// TwinCAT 3 PLC project plkV2
// ProgramVersion: 3.1.4024.0
// libraries:
//   Tc2_Standard, * (Beckhoff Automation GmbH)
//   Tc2_System, * (Beckhoff Automation GmbH)
//   Tc3_Module, * (Beckhoff Automation GmbH)
// project tree:
//   AUTOmovement/ A1.TcPOU, grab.TcPOU, moveCCW.TcPOU, moveCW.TcPOU, moveDown.TcPOU, moveIN.TcPOU, moveOUT.TcPOU, moveUP.TcPOU, relise.TcPOU
//   EdgeDetection/ EdgeDetection.TcPOU
//   / getBreadFromSensors.TcPOU, PlcTask.TcTTO
//   GVLs/ GVL.TcGVL, HMI.TcGVL
//   Muliplex/ Multiplexer.TcPOU
//   POUs/Automatic/ Automatic.TcPOU, AutomaticFB.TcPOU, FirstMove.TcPOU, SortTest.TcPOU, startSorting.TcPOU
//   POUs/ MAIN.TcPOU, MasterControl.TcPOU
//   POUs/Manual/ Manual.TcPOU
//   Timer/ AUTOtimer.TcPOU, TIMER.TcPOU

CONFIGURATION plkV2
    RESOURCE PLC ON TwinCAT3
        TASK PlcTask(INTERVAL := T#10ms, PRIORITY := 20);
        PROGRAM MasterControl WITH PlcTask : MasterControl;
    END_RESOURCE
END_CONFIGURATION

// ---- GVLs/GVL.TcGVL
{attribute 'qualified_only'}
VAR_GLOBAL
	//Automatic/manual
	ToggleSwitch AT %I* : BOOL; //0 - automatic; 1 - manual
	
	//lights
	LEDRed AT %Q* : BOOL; 
	LEDGreen AT %Q* : BOOL; 
	LEDupperBlue AT %Q* : BOOL; 
	LEDdownBlue AT %Q* : BOOL; 
	
	//buttons
	//upper
	ULBButton AT %I* : BOOL;
	URBButton AT %I* : BOOL;
	//lover
	LLBButton AT %I* : BOOL;
	LRBButton AT %I* : BOOL;
	//color
	GButton AT %I* : BOOL;
	RButton AT %I* : BOOL;


	//MOVESET
	//MoveUp/Down
	riseWay AT %Q* : BOOL; //0 - down, 1 - up
	riseAction AT %Q* : BOOL;
	
	
	//Rotation
	rotationWay AT %Q* : BOOL; //0 - CW, 1 - CCW
	rotationAction AT %Q* : BOOL;
	
	
	//Stretch
	stretchWay AT %Q* : BOOL; //0 - stretch, 1 - shrink
	stretchAction AT %Q* : BOOL;
	
	//claw
	clawWay AT %Q* : BOOL; //0 - open, 1 - release
	clawAction AT %Q* : BOOL;
	
	
	//SWITCHES
	//rotation
	SWrotation AT %I* : BOOL;
	SWstepsRotation AT %I* : BOOL;
	
	//stretch
	SWstretch AT %I* : BOOL;
	SWstepsStretch AT %I* : BOOL;
	
	//rise
	SWrise AT %I* : BOOL;
	SWstepsRise AT %I* : BOOL;
	
	//grab
	SWgrab AT %I* : BOOL;
	SWstepsGrab AT %I* : BOOL;
	
	
	//Bakery
	weight: REAL; //light - bagel, medium - toast/rye, heavy - baguette (weight sensor - HX711)
	color: INT; //white/black (color sensor - TCS3472)
	breadType: INT; //toast = 0; baguette = 1; rye = 2; bagel = 3
	binNumber: INT; // 2 or 4
	binFull: BOOL; //HC-SR04 x 2 or 4
	breadInfo : STRING; // white toast, white beguette, dark rye, dark bagel
	
	//objekt za pekarno - za HMI
	{attribute 'TcHmiSymbol'}
	BreadInfoID : INT := 0;
	
	
	{attribute 'TcHmiSymbol'}
	BinFullNumber : INT := 0;
	
	
	//nove lastnosti za senzorje
	breadColor : INT;
    breadWeightClass : STRING(10);
	breadID: INT;
	
 	{attribute 'TcHmiSymbol'}
	breadIDinfo : INT := 0;
	{attribute 'TcHmiSymbol'}
	breadIDText : STRING(10) := '';

    fullBin : INT;
	
	
	//za posodabljat koliko elementov je v škatli
	{attribute 'TcHmiSymbol'}
	BinUpdateTrigger : INT := 0;
	
	
	{attribute 'TcHmiSymbol'}
	breadTypeImageID : INT := 0; // 0=none, 1=toast, 2=baguette, 3=rye, 4=bagel
	//Sensors
	//BinIsFull : BOOL := FALSE;
	BinIsFull : INT := 0;	
	{attribute 'TcHmiSymbol'} Bin1Full : BOOL := FALSE;
	{attribute 'TcHmiSymbol'} Bin2Full : BOOL := FALSE;
	{attribute 'TcHmiSymbol'} Bin3Full : BOOL := FALSE;
	{attribute 'TcHmiSymbol'} Bin4Full : BOOL := FALSE;
	
	//breadColor: white, black
	{attribute 'TcHmiSymbol'}
	//breadColor : STRING(10) := 'NONE';
	
	
	//Number of bread in bin
    numToast   : INT := 0;
    numBaguette: INT := 0;
    numRye     : INT := 0;
    numBagel   : INT := 0;
	
	//STEVCI
	UniversalStevec AT %I* : BOOL;
	stevecGor AT %I* : BOOL;
	stevecRotacija AT %I* : BOOL;
	stevecSkrci AT %I* : BOOL;
	stevecKlesce AT %I* : BOOL;
	
	height AT %I* : REAL;
	rotation AT %I* : REAL;
	length AT %I* : REAL;
	grabMeter AT %I* : REAL;
	
	
	// AVTOMATIK PREMIKI
	upDone AT %Q* : BOOL;
	downDone AT %Q* : BOOL;
	CWDone AT %Q* : BOOL;
	CCWDone AT %Q* : BOOL;
	skrciDone AT %Q* : BOOL;
	raztegniDone AT %Q* : BOOL;
	grabDone AT %Q* : BOOL;
	reliseDone AT %Q* : BOOL;
	
	//GOR DOL
	gor AT %Q* : BOOL;
	dol AT %Q* : BOOL;
	
	//LEVO DESNO
	CW AT %Q* : BOOL;
	CCW AT %Q* : BOOL;
	
	//KLEŠČE--NE DELA!!!!
	primi AT %Q* : BOOL;
	spusti AT %Q* : BOOL;
	
	//IZTEG--NE DELA!!!!
	raztegniNaprej AT %Q* : BOOL;
	skrci AT %Q* : BOOL;
	
	
	//on/off
	isON AT %I* : BOOL;
END_VAR

// ---- GVLs/HMI.TcGVL
{attribute 'qualified_only'}
VAR_GLOBAL
	BreadIDpicked:INT;
	test:BOOL := FALSE;
	Action1:BOOL;
	Action2:BOOL;
END_VAR

// ---- POUs/MasterControl.TcPOU
PROGRAM MasterControl
VAR
	//preveri če je switvh aktiven
	Rocno: Manual;
	Avtomatik: Automatic;
	{attribute 'TcHmiSymbol'}
	premikanje: SortTest;

	
	
	Motor: BOOL;
	IS_Manual: BOOL;
	
	// Nova instanca za vrednotenje kruha
	BreadEval: getBreadFromSensors;
	
END_VAR

IS_Manual := GVL.ToggleSwitch;
IF IS_Manual THEN
	Rocno();
	//GVL.riseWay := Rocno.smer1;//asign GVL.way
ELSE
		//Avtomatik();
		premikanje();
END_IF

// Neodvisno od ročnega/avtomatskega režima – vedno preveri kruh
BreadEval(
	breadColor := GVL.breadColor,
	breadWeightClass := GVL.breadWeightClass
);

// Rezultat zapiši v GVL za HMI uporabo
GVL.breadTypeImageID := BreadEval.breadTypeImageID;
GVL.breadInfo := BreadEval.breadInfo;

END_PROGRAM

// ---- POUs/Manual/Manual.TcPOU
FUNCTION_BLOCK Manual
VAR_INPUT
END_VAR

VAR_OUTPUT
END_VAR

VAR
	motorSelect: Multiplexer;
	EdgeDetectionRedButton: EdgeDetection;
	TIMER: TIMER;
	
	CountDown: CTUD;
	EdgeDetectionCD: BOOL;
	dropTimer: TON;
	rotateTimer: TON;
	stretchTimer: TON;
	clawTimer: TON;
	CounterDol: CTUD;
	visina: WORD;
	CounterCCW: CTUD;
	rotacija: WORD;
	CounterRazteg: CTUD;
	dolzina: WORD;
	CounterKlesce: CTUD;
	prijem: WORD;
	CounterVisina: CTUD;
END_VAR

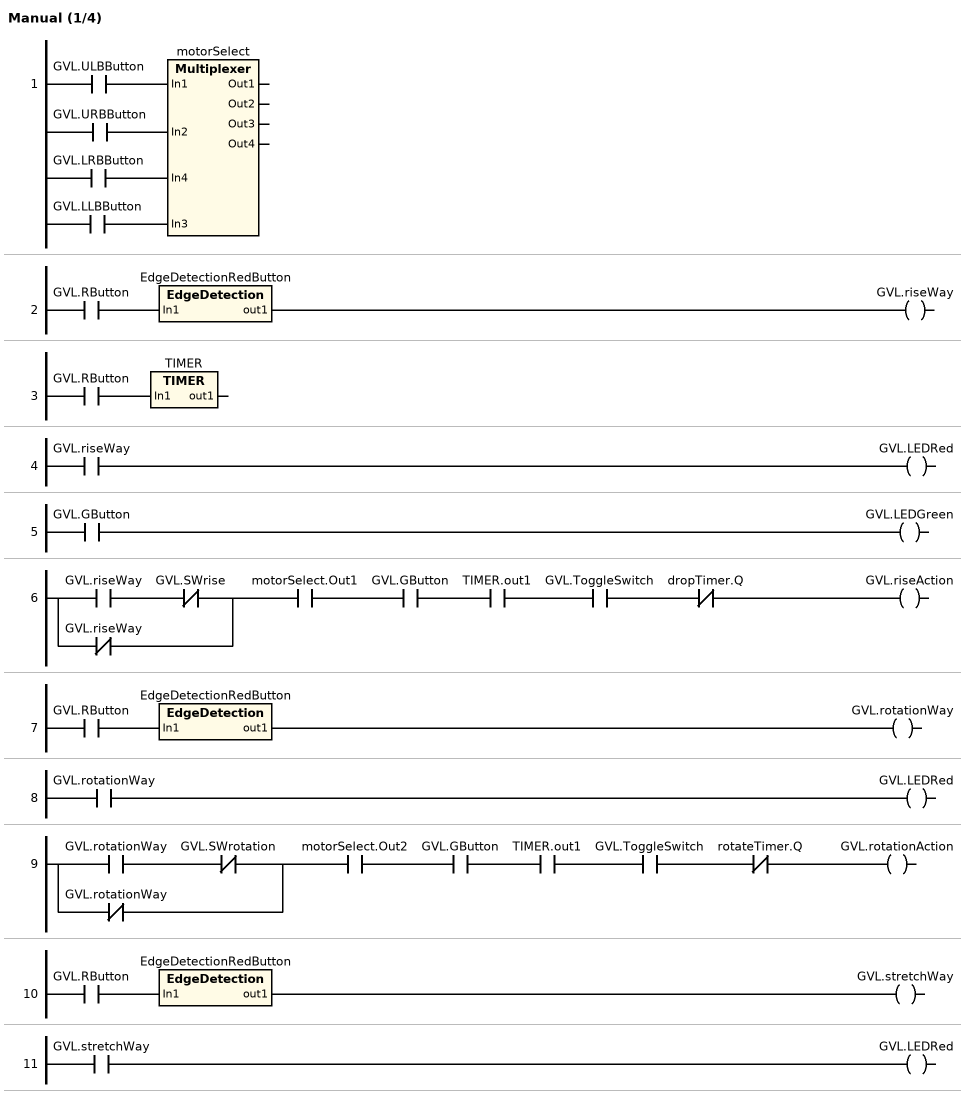
// NETWORK 1
motorSelect(In1 := GVL.ULBButton, In2 := GVL.URBButton, In4 := GVL.LRBButton, In3 := GVL.LLBButton); // Multiplexer

// NETWORK 2
EdgeDetectionRedButton(In1 := GVL.RButton); // EdgeDetection
GVL.riseWay := EdgeDetectionRedButton.out1;

// NETWORK 3
TIMER(In1 := GVL.RButton);

// NETWORK 4
GVL.LEDRed := GVL.riseWay;

// NETWORK 5
GVL.LEDGreen := GVL.GButton;

// NETWORK 6
GVL.riseAction := (GVL.riseWay AND NOT GVL.SWrise OR NOT GVL.riseWay) AND motorSelect.Out1 AND GVL.GButton AND TIMER.out1 AND GVL.ToggleSwitch AND NOT dropTimer.Q;

// NETWORK 7
EdgeDetectionRedButton(In1 := GVL.RButton); // EdgeDetection
GVL.rotationWay := EdgeDetectionRedButton.out1;

// NETWORK 8
GVL.LEDRed := GVL.rotationWay;

// NETWORK 9
GVL.rotationAction := (GVL.rotationWay AND NOT GVL.SWrotation OR NOT GVL.rotationWay) AND motorSelect.Out2 AND GVL.GButton AND TIMER.out1 AND GVL.ToggleSwitch AND NOT rotateTimer.Q;

// NETWORK 10
EdgeDetectionRedButton(In1 := GVL.RButton); // EdgeDetection
GVL.stretchWay := EdgeDetectionRedButton.out1;

// NETWORK 11
GVL.LEDRed := GVL.stretchWay;

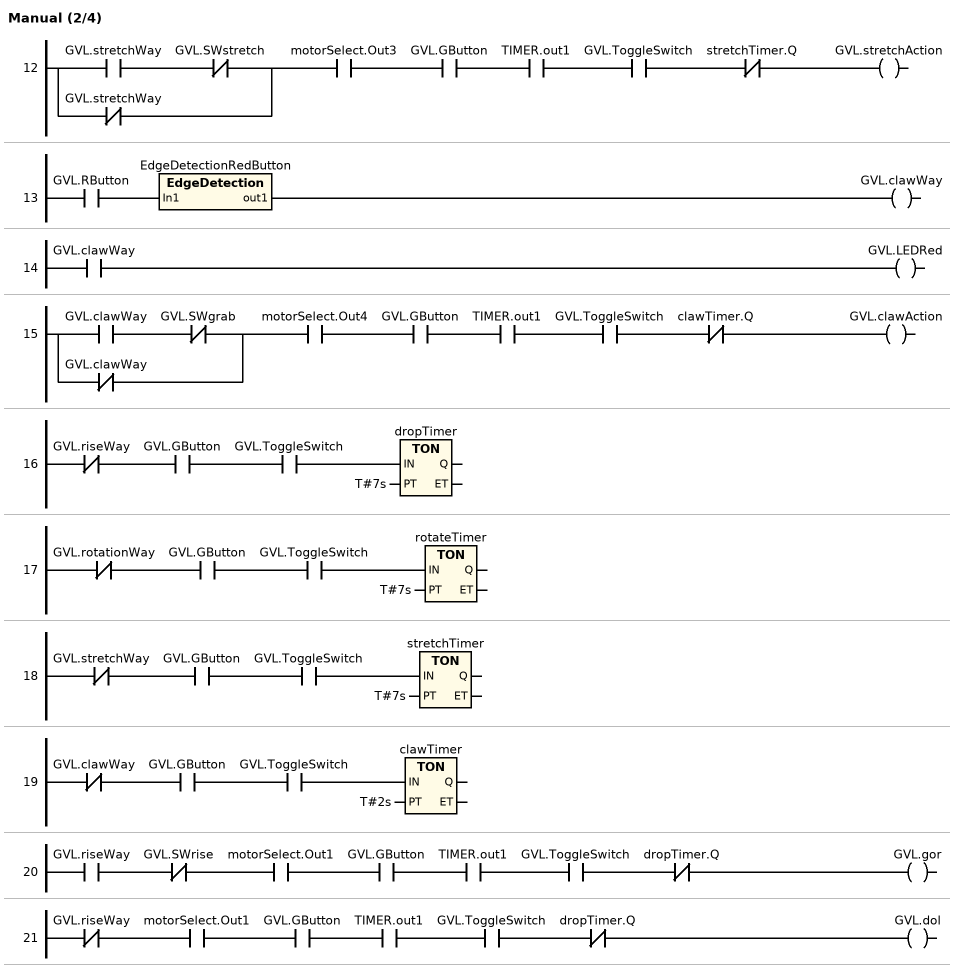
// NETWORK 12
GVL.stretchAction := (GVL.stretchWay AND NOT GVL.SWstretch OR NOT GVL.stretchWay) AND motorSelect.Out3 AND GVL.GButton AND TIMER.out1 AND GVL.ToggleSwitch AND NOT stretchTimer.Q;

// NETWORK 13
EdgeDetectionRedButton(In1 := GVL.RButton); // EdgeDetection
GVL.clawWay := EdgeDetectionRedButton.out1;

// NETWORK 14
GVL.LEDRed := GVL.clawWay;

// NETWORK 15
GVL.clawAction := (GVL.clawWay AND NOT GVL.SWgrab OR NOT GVL.clawWay) AND motorSelect.Out4 AND GVL.GButton AND TIMER.out1 AND GVL.ToggleSwitch AND NOT clawTimer.Q;

// NETWORK 16
dropTimer(IN := NOT GVL.riseWay AND GVL.GButton AND GVL.ToggleSwitch, PT := T#7s); // TON

// NETWORK 17
rotateTimer(IN := NOT GVL.rotationWay AND GVL.GButton AND GVL.ToggleSwitch, PT := T#7s); // TON

// NETWORK 18
stretchTimer(IN := NOT GVL.stretchWay AND GVL.GButton AND GVL.ToggleSwitch, PT := T#7s); // TON

// NETWORK 19
clawTimer(IN := NOT GVL.clawWay AND GVL.GButton AND GVL.ToggleSwitch, PT := T#2s); // TON

// NETWORK 20
GVL.gor := GVL.riseWay AND NOT GVL.SWrise AND motorSelect.Out1 AND GVL.GButton AND TIMER.out1 AND GVL.ToggleSwitch AND NOT dropTimer.Q;

// NETWORK 21
GVL.dol := NOT GVL.riseWay AND motorSelect.Out1 AND GVL.GButton AND TIMER.out1 AND GVL.ToggleSwitch AND NOT dropTimer.Q;

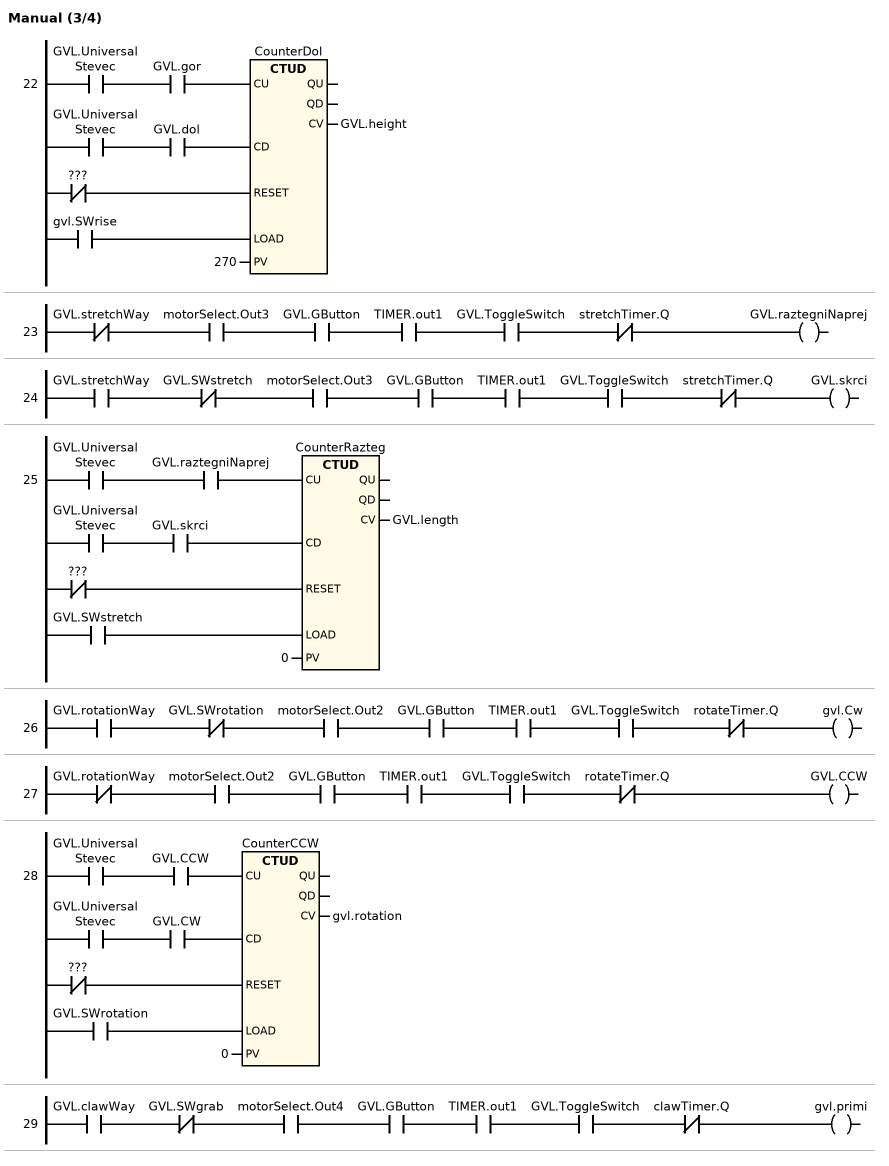
// NETWORK 22
CounterDol(
    CU := GVL.UniversalStevec AND GVL.gor,
    CD := GVL.UniversalStevec AND GVL.dol,
    LOAD := gvl.SWrise,
    PV := 270,
    CV => GVL.height); // CTUD

// NETWORK 23
GVL.raztegniNaprej := NOT GVL.stretchWay AND motorSelect.Out3 AND GVL.GButton AND TIMER.out1 AND GVL.ToggleSwitch AND NOT stretchTimer.Q;

// NETWORK 24
GVL.skrci := GVL.stretchWay AND NOT GVL.SWstretch AND motorSelect.Out3 AND GVL.GButton AND TIMER.out1 AND GVL.ToggleSwitch AND NOT stretchTimer.Q;

// NETWORK 25
CounterRazteg(
    CU := GVL.UniversalStevec AND GVL.raztegniNaprej,
    CD := GVL.UniversalStevec AND GVL.skrci,
    LOAD := GVL.SWstretch,
    PV := 0,
    CV => GVL.length); // CTUD

// NETWORK 26
gvl.Cw := GVL.rotationWay AND NOT GVL.SWrotation AND motorSelect.Out2 AND GVL.GButton AND TIMER.out1 AND GVL.ToggleSwitch AND NOT rotateTimer.Q;

// NETWORK 27
GVL.CCW := NOT GVL.rotationWay AND motorSelect.Out2 AND GVL.GButton AND TIMER.out1 AND GVL.ToggleSwitch AND NOT rotateTimer.Q;

// NETWORK 28
CounterCCW(
    CU := GVL.UniversalStevec AND GVL.CCW,
    CD := GVL.UniversalStevec AND GVL.CW,
    LOAD := GVL.SWrotation,
    PV := 0,
    CV => gvl.rotation); // CTUD

// NETWORK 29
gvl.primi := GVL.clawWay AND NOT GVL.SWgrab AND motorSelect.Out4 AND GVL.GButton AND TIMER.out1 AND GVL.ToggleSwitch AND NOT clawTimer.Q;

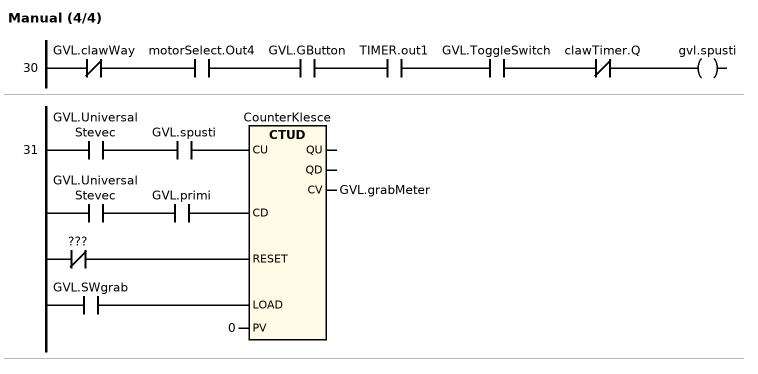
// NETWORK 30
gvl.spusti := NOT GVL.clawWay AND motorSelect.Out4 AND GVL.GButton AND TIMER.out1 AND GVL.ToggleSwitch AND NOT clawTimer.Q;

// NETWORK 31
CounterKlesce(
    CU := GVL.UniversalStevec AND GVL.spusti,
    CD := GVL.UniversalStevec AND GVL.primi,
    LOAD := GVL.SWgrab,
    PV := 0,
    CV => GVL.grabMeter); // CTUD

END_FUNCTION_BLOCK

// ---- Muliplex/Multiplexer.TcPOU
FUNCTION_BLOCK Multiplexer
VAR_INPUT
	In1: BOOL;
	In2: BOOL;
	In4: BOOL;
	In3: BOOL;
END_VAR

VAR_OUTPUT
	Out1: BOOL;
	Out2: BOOL;
	Out3: BOOL;
	Out4: BOOL;
END_VAR

VAR
	UpDown: RS;
	CWCCW: RS;
	StretchShrink: RS;
	GrabRelease: RS;
END_VAR

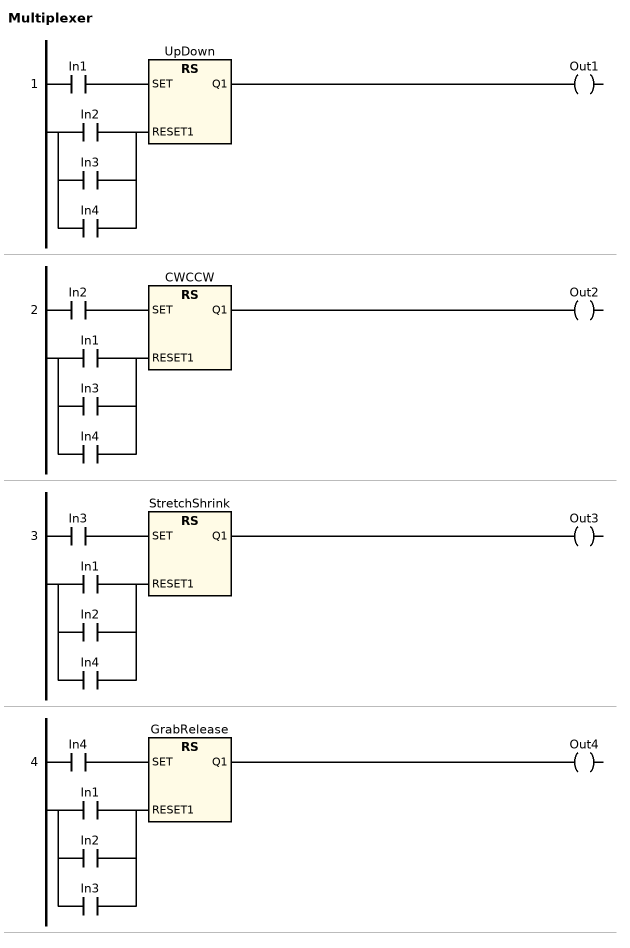
// NETWORK 1
UpDown(SET := In1, RESET1 := In2 OR In3 OR In4); // RS
Out1 := UpDown.Q1;

// NETWORK 2
CWCCW(SET := In2, RESET1 := In1 OR In3 OR In4); // RS
Out2 := CWCCW.Q1;

// NETWORK 3
StretchShrink(SET := In3, RESET1 := In1 OR In2 OR In4); // RS
Out3 := StretchShrink.Q1;

// NETWORK 4
GrabRelease(SET := In4, RESET1 := In1 OR In2 OR In3); // RS
Out4 := GrabRelease.Q1;

END_FUNCTION_BLOCK

// ---- EdgeDetection/EdgeDetection.TcPOU
FUNCTION_BLOCK EdgeDetection
VAR_INPUT
	In1: BOOL;
END_VAR
VAR_OUTPUT
	out1: BOOL;
END_VAR
VAR
	EdgeDetection1: R_TRIG;
	MemoryCell1: RS;
END_VAR

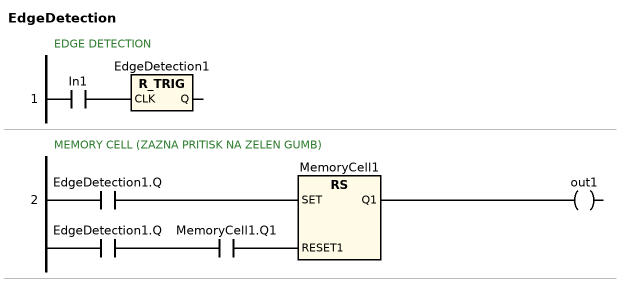
// NETWORK 1
// EDGE DETECTION
EdgeDetection1(CLK := In1); // R_TRIG

// NETWORK 2
// MEMORY CELL (ZAZNA PRITISK NA ZELEN GUMB)
MemoryCell1(SET := EdgeDetection1.Q, RESET1 := EdgeDetection1.Q AND MemoryCell1.Q1); // RS
out1 := MemoryCell1.Q1;

END_FUNCTION_BLOCK

// ---- Timer/TIMER.TcPOU
FUNCTION_BLOCK TIMER
VAR_INPUT
	In1: BOOL;
END_VAR
VAR_OUTPUT
	out1: BOOL;
END_VAR
VAR
	Timer1: TON;
	ontValue: TIME;
END_VAR

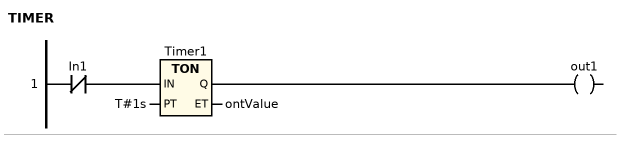
// NETWORK 1
Timer1(IN := NOT In1, PT := T#1s, ET => ontValue); // TON
out1 := Timer1.Q;

END_FUNCTION_BLOCK

// ---- POUs/Automatic/Automatic.TcPOU
FUNCTION_BLOCK Automatic
VAR_INPUT	
END_VAR
VAR_OUTPUT
END_VAR
VAR
    R1 : FirstMove;
    previousBreadID : INT := 0;
	i : INT := 1;
    triggerStart : BOOL := FALSE;
    isRunning : BOOL := FALSE;
END_VAR

// Če kruh še ni v obdelavi in pride nov breadID
//IF NOT isRunning AND GVL.breadID <> 0 AND GVL.breadID <> previousBreadID THEN
IF NOT isRunning AND GVL.breadID <> 0 THEN
	R1.itemID := GVL.breadID; // Nastavi novi kruh
	triggerStart := TRUE;
	previousBreadID := GVL.breadID; // Posodobi si trenutno vrednost
END_IF

// Poženi sekvenco, če je bil sprožen nov klic
IF triggerStart THEN
	R1(); // Pokliči FB
	isRunning := TRUE;
END_IF

// Nadaljuj izvajanje sekvence
IF isRunning THEN
	R1(); // Sekvenca se še izvaja
   IF R1.done THEN
		isRunning := FALSE;
		GVL.breadID := 0;           // Reset za TwinCAT
		previousBreadID := 0;       // Omogoči, da tudi isti kruh lahko pride ponovno
		triggerStart := FALSE;      // Reset sprožilca
	END_IF
END_IF

END_FUNCTION_BLOCK

// ---- POUs/Automatic/FirstMove.TcPOU
FUNCTION_BLOCK FirstMove
VAR_INPUT
    grab: grab; 
	timer : TP;	
	ccw: moveCCW;
	cw:moveCW;
	down:moveDown;
	iztegni:moveOUT;
	skrci:moveIN;
	up: moveUp;
	relise: relise; 
	itemID: INT := GVL.breadID;
END_VAR
VAR_OUTPUT
	 done: BOOL := FALSE; // Indikator, da je sekvenca zaključena
END_VAR
VAR
	currentState: INT := 0; // Trenutno stanje sekvence
	
	obDol: INT;
	objekt: INT;
	//itemID: INT := 1; //item number
	
	TimerWait: TOF;
	I: INT;
END_VAR

CASE currentState OF
	
	0:
		done := FALSE;
		GVL.downDone := FALSE;
		GVL.grabDone := FALSE;
		currentState := 1;
	
	1:
		down(seconds := T#5S);  // Aktiviraj premik dol
		IF GVL.downDone THEN          // Počakaj, da je premik zaključen
			currentState := 2;     // Premik na naslednje stanje
			GVL.downDone := FALSE;
		END_IF
		
	2:
		grab(seconds := T#2.2S);
		IF GVL.grabDone THEN           // Počakaj, da je prijem zaključen
			currentState := 3;      // Premik na naslednje stanje
			GVL.grabDone := FALSE;
		END_IF
		
	3:
		up(seconds := T#7S);
        IF GVL.upDone THEN           // Počakaj, da je prijem zaključen
            currentState := 4;      // Premik na naslednje stanje
			GVL.upDone := FALSE;
        END_IF

	4:
		//bageta
		IF itemID = 1 THEN
			cw(seconds := T#1.9S);
			IF GVL.CWDone THEN           // Počakaj, da je prijem zaključen
				currentState := 5;      // Premik na naslednje stanje
				GVL.CWDone := FALSE;
			END_IF
		//toast
		ELSIF itemID = 2 THEN
			cw(seconds := T#2.6S);
			IF GVL.CWDone THEN           // Počakaj, da je prijem zaključen
				currentState := 5;      // Premik na naslednje stanje
				GVL.CWDone := FALSE;
			END_IF
		//rženi kruh
		ELSIF itemID = 3 THEN
			cw(seconds := T#3.7S);
			IF GVL.CWDone THEN           // Počakaj, da je prijem zaključen
				currentState := 5;      // Premik na naslednje stanje
				GVL.CWDone := FALSE;
			END_IF
		//bagel
		ELSIF itemID = 4 THEN
			cw(seconds := T#4.2S);
			IF GVL.CWDone THEN           // Počakaj, da je prijem zaključen
				currentState := 5;      // Premik na naslednje stanje
				GVL.CWDone := FALSE;
			END_IF
		END_IF
		
	
	5:
	IF itemID = 1 THEN
		iztegni(seconds := T#4S);
        IF GVL.skrciDone THEN           // Počakaj, da je prijem zaključen
            currentState := 6;      // Premik na naslednje stanje
			GVL.skrciDone := FALSE;
        END_IF
	ELSIF itemID = 2 THEN
		iztegni(seconds := T#2.3S);
        IF GVL.skrciDone THEN           // Počakaj, da je prijem zaključen
            currentState := 6;      // Premik na naslednje stanje
			GVL.skrciDone := FALSE;
        END_IF
	ELSIF itemID = 3 THEN				
		iztegni(seconds := T#2.3S);
        IF GVL.skrciDone THEN           // Počakaj, da je prijem zaključen
            currentState := 6;      // Premik na naslednje stanje
			GVL.skrciDone := FALSE;
        END_IF
	ELSIF itemID = 4 THEN
		iztegni(seconds := T#4.3S);
        IF GVL.skrciDone THEN           // Počakaj, da je prijem zaključen
            currentState := 6;      // Premik na naslednje stanje
			GVL.skrciDone := FALSE;
        END_IF
	END_IF
		
	
	6:
		relise(seconds := T#3S);
        IF GVL.reliseDone THEN           // Počakaj, da je prijem zaključen
            currentState := 7;      // Premik na naslednje stanje
			GVL.reliseDone := FALSE;
        END_IF
	
	7:
		skrci(seconds := T#6S);
        IF GVL.skrciDone THEN           // Počakaj, da je prijem zaključen
            currentState := 8;      // Premik na naslednje stanje
			GVL.skrciDone := FALSE;
        END_IF
	
	8:
		ccw(seconds := T#6S);
        IF GVL.CWDone THEN           // Počakaj, da je prijem zaključen
            //currentState := 9;      // Premik na naslednje stanje
			currentState := 9;
			GVL.CWDone := FALSE;
        END_IF
		
	//9:
	//	GVL.upDone := FALSE;
	//	up(seconds := T#7S);
    //    IF GVL.upDone THEN           // Počakaj, da je prijem zaključen
    //        currentState := 0;      // Premik na naslednje stanje
	//		GVL.upDone := FALSE;
    //    END_IF
	
	 9:
        done := TRUE;               // Označi, da je sekvenca zaključena
        currentState := 0;          // Ponastavi na začetno stanje

	 
END_CASE

END_FUNCTION_BLOCK

// ---- AUTOmovement/grab.TcPOU
FUNCTION_BLOCK grab
VAR_INPUT
	 seconds: TIME; //time of moving	  
END_VAR
VAR_OUTPUT
	done: BOOL := FALSE; // output of finished work
END_VAR
VAR
	TimerNewGrab: AUTOtimer;
	activated: BOOL := FALSE; // Internal logic for activation
	grabEnd: BOOL := FALSE;
END_VAR

IF NOT activated THEN
    TimerNewGrab(vrednost := TRUE, inpCas := seconds, outCas => grabEnd);
    activated := TRUE;
END_IF

IF grabEnd  THEN
    TimerNewGrab(vrednost := FALSE, inpCas := seconds, outCas => grabEnd);
	GVL.primi := TRUE;
	GVL.clawWay := FALSE;
    GVL.clawAction := TRUE;  // grab active 
    GVL.grabDone := FALSE; // The move is not finished yet
	GVL.grabMeter := GVL.grabMeter + 0.4;
ELSE
	GVL.primi  := FALSE;
	GVL.clawWay := FALSE;
    GVL.clawAction := FALSE;     // Stop grabing
    GVL.grabDone:= TRUE;  // Mark the end of the move
	activated := FALSE;
END_IF

END_FUNCTION_BLOCK

// ---- Timer/AUTOtimer.TcPOU
FUNCTION_BLOCK AUTOtimer
VAR_INPUT
	vrednost: BOOL;
	inpCas: TIME;
END_VAR
VAR_OUTPUT
	outCas: BOOL;
END_VAR
VAR
	TimerAutomatic: TOF;
END_VAR

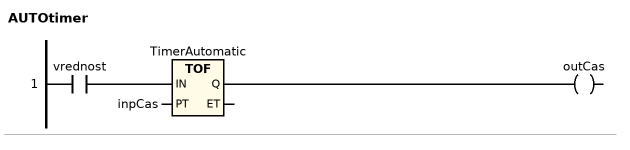
// NETWORK 1
TimerAutomatic(IN := vrednost, PT := inpCas); // TOF
outCas := TimerAutomatic.Q;

END_FUNCTION_BLOCK

// ---- AUTOmovement/moveCCW.TcPOU
FUNCTION_BLOCK moveCCW
VAR_INPUT
	 seconds: TIME;  //time of moving
END_VAR
VAR_OUTPUT
	 done: BOOL := FALSE; // output of finished work
END_VAR
VAR
	TimerNewCCW: AUTOtimer; 
	activated: BOOL := FALSE; // Internal logic for activation
	CCWend: BOOL := FALSE;
END_VAR

IF NOT activated THEN
    TimerNewCCW(vrednost := TRUE, inpCas := seconds, outCas => CCWend);
    activated := TRUE;
END_IF

IF CCWend AND NOT GVL.SWrotation THEN
    TimerNewCCW(vrednost := FALSE, inpCas := seconds, outCas => CCWend);
	GVL.CCW := TRUE;
    GVL.rotationWay := TRUE;      
	GVL.rotationAction := TRUE;  // CCW active 
  	GVL.CCWDone := FALSE;    // The move is not finished yet
	GVL.rotation := GVL.rotation - 0.5;
ELSE
	GVL.CCW := FALSE; 
   	GVL.rotationWay := FALSE;      
	GVL.rotationAction := FALSE;    // Stop moving CCW
   	GVL.CCWDone := TRUE;   // Mark the end of the move
	activated := FALSE;
END_IF

END_FUNCTION_BLOCK

// ---- AUTOmovement/moveCW.TcPOU
FUNCTION_BLOCK moveCW
VAR_INPUT
	seconds: TIME; //time of moving
END_VAR
VAR_OUTPUT
	 done: BOOL := FALSE; // output of finished work
END_VAR
VAR
	TimerNewCW: AUTOtimer;
	activated: BOOL := FALSE; // Internal logic for activation
	CWend: BOOL := FALSE;
END_VAR

IF NOT activated THEN
    TimerNewCW(vrednost := TRUE, inpCas := seconds, outCas => CWend);
    activated := TRUE;
END_IF

IF CWend THEN
    TimerNewCW(vrednost := FALSE, inpCas := seconds, outCas => CWend);
	GVL.CW := TRUE; 
    GVL.rotationWay := FALSE; 
	GVL.rotationAction := TRUE;  // CCW active 
  	GVL.CWDone := FALSE;     // The move is not finished yet
	GVL.rotation := GVL.rotation + 0.5;
ELSE
	GVL.CW := FALSE;
   	GVL.rotationWay := FALSE; 
	GVL.rotationAction := FALSE;        // Stop moving CW
    GVL.CWDone := TRUE;    // Mark the end of the move
	//CWend := FALSE;
	activated := FALSE;
END_IF

END_FUNCTION_BLOCK

// ---- AUTOmovement/moveDown.TcPOU
FUNCTION_BLOCK moveDown
VAR_INPUT
	seconds: TIME; //time of moving
END_VAR
VAR_OUTPUT
	done: BOOL := FALSE;  // output of finished work
END_VAR
VAR
	TimerNewDown: AUTOtimer; 
	aktiviran: BOOL := FALSE; // Internal logic for activation
	DownEnd: BOOL := FALSE;
END_VAR

IF NOT aktiviran THEN
    TimerNewDown(vrednost := TRUE, inpCas := seconds, outCas => DownEnd);
    aktiviran := TRUE;
END_IF

IF DownEnd THEN
    TimerNewDown(vrednost := FALSE, inpCas := seconds, outCas => DownEnd);
	GVL.dol := TRUE;
	GVL.riseWay := FALSE;
	GVL.riseAction := TRUE; 	// down active 
  	GVL.downDone := FALSE;    // The move is not finished yet
	GVL.height := GVL.height - 0.4;
ELSE
	GVL.dol := FALSE;
   	GVL.riseWay := FALSE;
	GVL.riseAction := FALSE;	// Stop moving down
   	GVL.downDone := TRUE;   // Mark the end of the move
	aktiviran := FALSE;
END_IF

END_FUNCTION_BLOCK

// ---- AUTOmovement/moveOUT.TcPOU
FUNCTION_BLOCK moveOUT
VAR_INPUT
    seconds: TIME;     //time of moving
END_VAR

VAR_OUTPUT
    done: BOOL := FALSE; // output of finished work
END_VAR

VAR
	TimerNewOUT: AUTOtimer;
	activated: BOOL := FALSE; // Internal logic for activation
	OUTend: BOOL := FALSE;
END_VAR

IF NOT activated THEN
    TimerNewOUT(vrednost := TRUE, inpCas := seconds, outCas => OUTend);
    activated := TRUE;
END_IF

IF OUTend THEN //check switch aswell
    TimerNewOUT(vrednost := FALSE, inpCas := seconds, outCas => OUTend);
   	GVL.raztegniNaprej := TRUE;
	GVL.stretchWay := FALSE; 
	GVL.stretchAction := TRUE;      // shrink active
    GVL.skrciDone := FALSE;    // Označi zaključek premika
	GVL.length := GVL.length + 0.45;
ELSE
	GVL.raztegniNaprej := FALSE;
   	GVL.stretchWay := TRUE; 
	GVL.stretchAction := FALSE;        // Stop shrinking
    GVL.skrciDone := TRUE;   // Mark the end of the move
	activated := FALSE;
END_IF

END_FUNCTION_BLOCK

// ---- AUTOmovement/moveIN.TcPOU
FUNCTION_BLOCK moveIN
VAR_INPUT
    seconds: TIME;     //time of moving
END_VAR

VAR_OUTPUT
    done: BOOL := FALSE; // output of finished work
END_VAR

VAR
	TimerNewIN: AUTOtimer;
	activated: BOOL := FALSE; // Internal logic for activation
	INend: BOOL := FALSE;
END_VAR

IF NOT activated THEN
    TimerNewIN(vrednost := TRUE, inpCas := seconds, outCas => INend);
    activated := TRUE;
END_IF

IF INend AND NOT GVL.SWstretch THEN //check switch aswell
    TimerNewIN(vrednost := FALSE, inpCas := seconds, outCas => INend);
   	GVL.skrci := TRUE;
	GVL.stretchWay := TRUE; 
	GVL.stretchAction := TRUE;      // shrink active
    GVL.skrciDone := FALSE;    // Označi zaključek premika
	GVL.length := GVL.length - 0.5;
ELSE
	GVL.skrci := FALSE;
   	GVL.stretchWay := TRUE; 
	GVL.stretchAction := FALSE;        // Stop shrinking
    GVL.skrciDone := TRUE;   // Mark the end of the move
	activated := FALSE;
END_IF

END_FUNCTION_BLOCK

// ---- AUTOmovement/moveUP.TcPOU
FUNCTION_BLOCK moveUP
VAR_INPUT
	 seconds: TIME; //time of moving
END_VAR
VAR_OUTPUT
	done: BOOL := FALSE; // output of finished work
END_VAR
VAR
	TimerNewUP: AUTOtimer;
	activated: BOOL := FALSE; // Internal logic for activation
	UPend: BOOL := FALSE;
END_VAR


IF NOT activated THEN
    TimerNewUP(vrednost := TRUE, inpCas := seconds, outCas => UPend);
    activated := TRUE;
END_IF

IF UPend AND NOT GVL.SWrise THEN
    TimerNewUP(vrednost := FALSE, inpCas := seconds, outCas => UPend);
	GVL.gor := TRUE;  
	GVL.riseWay := TRUE;
	GVL.riseAction := TRUE;      // Ustavi premik gor
    GVL.upDone := FALSE;    // Označi zaključek premika
	GVL.height := GVL.height + 0.6;
ELSE
	GVL.gor := FALSE; 
    GVL.riseWay := FALSE;
	GVL.riseAction := FALSE;        // Premik gor aktiven
    GVL.upDone := TRUE;   // Premik še ni končan
	activated := FALSE;
END_IF

END_FUNCTION_BLOCK

// ---- AUTOmovement/relise.TcPOU
FUNCTION_BLOCK relise
VAR_INPUT
	 seconds: TIME; 
END_VAR
VAR_OUTPUT
	done: BOOL := FALSE;
END_VAR
VAR
	TimerNewRelise: AUTOtimer; // Trenutno pomemben
	aktiviran: BOOL := FALSE; // Notranja logika za aktivacijo
	KoncRelise: BOOL := FALSE;
END_VAR

IF NOT aktiviran THEN
    TimerNewRelise(vrednost := TRUE, inpCas := seconds, outCas => KoncRelise);
    aktiviran := TRUE;
END_IF

IF KoncRelise AND NOT GVL.SWgrab THEN
    TimerNewRelise(vrednost := FALSE, inpCas := seconds, outCas => KoncRelise);
	GVL.spusti := TRUE;
	GVL.clawWay := TRUE;
    GVL.clawAction := TRUE;     // Ustavi premik gor
  	GVL.reliseDone := FALSE;    // Označi zaključek premika
	GVL.grabMeter := GVL.grabMeter - 0.6;
ELSE
	GVL.spusti := FALSE;
   	GVL.clawWay := TRUE;
    GVL.clawAction := FALSE;      // Premik gor aktiven
   	GVL.reliseDone := TRUE;   // Premik še ni končan
	aktiviran := FALSE;
END_IF

END_FUNCTION_BLOCK

// ---- POUs/Automatic/SortTest.TcPOU
FUNCTION_BLOCK SortTest
VAR_INPUT
    grab: grab;
    timer: TP;
    ccw: moveCCW;
    cw: moveCW;
    down: moveDown;
    iztegni: moveOUT;
    skrci: moveIN;
    up: moveUp;
    relise: relise;
END_VAR

VAR_OUTPUT
    done: BOOL := FALSE;
END_VAR

VAR
    currentState: INT := 100; // Start at new state for waiting
  
	{attribute 'TcHmiSymbol'}
	//itemID: INT := 0;
	itemID: INT := 1;
    previousBreadID: INT := 0;
END_VAR

CASE currentState OF

    // 100 – Čakaj na nov objekt
    100:
        done := FALSE;
        IF GVL.breadID <> 0 AND GVL.breadID <> previousBreadID THEN
            itemID := GVL.breadID;
            GVL.BreadInfoID := itemID;
            GVL.breadID := 0; // Počistimo, da bo Arduino lahko poslal novega
            currentState := 0;
        END_IF

    // 0: Inicializacija
    0:
        GVL.downDone := FALSE;
        GVL.grabDone := FALSE;
        currentState := 1;

    // 1: Premik dol
    1:
        down(seconds := T#5S);
        IF GVL.downDone THEN
            GVL.downDone := FALSE;
            currentState := 2;
        END_IF

    // 2: Prijem
    2:
        grab(seconds := T#2.2S);
        IF GVL.grabDone THEN
            GVL.grabDone := FALSE;
            currentState := 3;
        END_IF

    // 3: Dvig
    3:
        up(seconds := T#7S);
        IF GVL.upDone THEN
            GVL.upDone := FALSE;
            currentState := 4;
        END_IF

    // 4: Rotacija CW glede na tip kruha
    4:
        CASE itemID OF
            1: cw(seconds := T#1.9S); // Bageta
            2: cw(seconds := T#2.6S); // Toast
            3: cw(seconds := T#3.7S); // Rženi
            4: cw(seconds := T#4.2S); // Bagel
        END_CASE
        IF GVL.CWDone THEN
            GVL.CWDone := FALSE;
            currentState := 5;
        END_IF

    // 5: Iztegni roko
    5:
        CASE itemID OF
            1: iztegni(seconds := T#4S);
            2: iztegni(seconds := T#2.3S);
            3: iztegni(seconds := T#2.3S);
            4: iztegni(seconds := T#4.3S);
        END_CASE
        IF GVL.skrciDone THEN
            GVL.skrciDone := FALSE;
            currentState := 6;
        END_IF

    // 6: Spusti kruh
    6:
        relise(seconds := T#3S);
        IF GVL.reliseDone THEN
            GVL.reliseDone := FALSE;
			//GVL.BinUpdateTrigger := itemID;
            currentState := 7;
        END_IF

    // 7: Roka se skrči nazaj
    7:
        skrci(seconds := T#6S);
        IF GVL.skrciDone THEN
            GVL.skrciDone := FALSE;
			//GVL.BinUpdateTrigger := 0;
            currentState := 8;
        END_IF

    // 8: Povratek z rotacijo CCW
    8:
        ccw(seconds := T#6S);
        IF GVL.CCWDone THEN
            GVL.CCWDone := FALSE;
            currentState := 9;
        END_IF

    // 9: Zaključi cikel
    9:
        done := TRUE;
        currentState := 100; // Vrni se na čakanje novega objekta
END_CASE

END_FUNCTION_BLOCK

// ---- getBreadFromSensors.TcPOU
FUNCTION_BLOCK getBreadFromSensors
VAR_INPUT
	breadColor: INT;
	breadWeightClass: STRING;
END_VAR
VAR_OUTPUT
	breadTypeImageID: INT;
	breadInfo: STRING;
END_VAR
VAR	
END_VAR

IF breadColor = 0 AND breadWeightClass = 'medium' THEN
    breadTypeImageID := 1; // Toast
    breadInfo := 'White Toast';
ELSIF breadColor = 0 AND breadWeightClass = 'heavy' THEN
    breadTypeImageID := 2; // Baguette
    breadInfo := 'White Baguette';
ELSIF breadColor = 1 AND breadWeightClass = 'medium' THEN
    breadTypeImageID := 3; // Rye
    breadInfo := 'Dark Rye';
ELSIF breadColor = 1 AND breadWeightClass = 'light' THEN
    breadTypeImageID := 4; // Bagel
    breadInfo := 'Dark Bagel';
ELSE
    breadTypeImageID := 0;
    breadInfo := 'Unknown';
END_IF;

END_FUNCTION_BLOCK

// ---- AUTOmovement/A1.TcPOU
FUNCTION_BLOCK A1
VAR_INPUT
END_VAR
VAR_OUTPUT
END_VAR
VAR
	R1: Recepie1;
	stateReset: INT := 1;
END_VAR

IF stateReset = 0 THEN
	R1();
END_IF

RETURN;

END_FUNCTION_BLOCK

// ---- POUs/Automatic/AutomaticFB.TcPOU
FUNCTION_BLOCK AutomaticFB
VAR_INPUT
END_VAR
VAR_OUTPUT
END_VAR
VAR
END_VAR

// NETWORK 1

END_FUNCTION_BLOCK

// ---- POUs/Automatic/startSorting.TcPOU
FUNCTION_BLOCK startSorting
VAR_INPUT
    grab: grab; 
	timer : TP;	
	ccw: moveCCW;
	cw:moveCW;
	down:moveDown;
	iztegni:moveOUT;
	skrci:moveIN;
	up: moveUp;
	relise: relise; 
END_VAR
VAR_OUTPUT
	 done: BOOL := FALSE; // Indikator, da je sekvenca zaključena
END_VAR
VAR
	currentState: INT := 0; // Trenutno stanje sekvence
	
	obDol: INT;
	objekt: INT;
	itemID: INT := 1; //item number
	TimerWait: TOF;
	I: INT;
END_VAR

CASE currentState OF
    // Stanje 0: Priprava
    0:
        done := FALSE;         // Ponastavi indikator zaključka
        GVL.downDone := FALSE;     // Ponastavi zastavico za premik dol
        GVL.grabDone := FALSE;     // Ponastavi zastavico za prijem
        currentState := 1;     // Premik na naslednje stanje

    1://PREMIK DOL PO OBJEKTIH
		 //grab(seconds := T#1.5S);     // Aktiviraj prijem
		grab(seconds := T#2.2S);
        IF GVL.grabDone THEN           // Počakaj, da je prijem zaključen
            //grabDone := TRUE;       // Nastavi zastavico
            currentState := 2;      // Premik na naslednje stanje
			GVL.grabDone := FALSE;
        END_IF
		
	2:	
		ccw(seconds := T#2.5S);
			IF GVL.CCWDone THEN           // Počakaj, da je prijem zaključen
				currentState := 3;      // Premik na naslednje stanje
				GVL.CCWDone := FALSE;
			END_IF
			
	3:
		cw(seconds := T#2.5S);
        IF GVL.CWDone THEN           // Počakaj, da je prijem zaključen
            currentState := 4;      // Premik na naslednje stanje
			GVL.CWDone := FALSE;
        END_IF
	4:
		down(seconds := T#1S);  // Aktiviraj premik dol
		IF GVL.downDone THEN          // Počakaj, da je premik zaključen
			//downDone := TRUE;      // Nastavi zastavico
			currentState := 5;     // Premik na naslednje stanje
			GVL.downDone := FALSE;
		END_IF
		
	5:
		iztegni(seconds := T#1S);
        IF GVL.skrciDone THEN           // Počakaj, da je prijem zaključen
            currentState := 6;      // Premik na naslednje stanje
			GVL.skrciDone := FALSE;
        END_IF
		
	6:
		skrci(seconds := T#1S);
        IF GVL.skrciDone THEN           // Počakaj, da je prijem zaključen
            currentState := 7;      // Premik na naslednje stanje
			GVL.skrciDone := FALSE;
        END_IF
	7:
		up(seconds := T#2S);
        IF GVL.upDone THEN           // Počakaj, da je prijem zaključen
            currentState := 8;      // Premik na naslednje stanje
			GVL.upDone := FALSE;
        END_IF
	8:
		relise(seconds := T#2S);
        IF GVL.reliseDone THEN           // Počakaj, da je prijem zaključen
            currentState := 8;      // Premik na naslednje stanje
			GVL.reliseDone := FALSE;
        END_IF
	
END_CASE

END_FUNCTION_BLOCK

// ---- POUs/MAIN.TcPOU
PROGRAM MAIN
VAR
END_VAR

END_PROGRAM
